FUNCTION_BLOCK FB_Pomp IMPLEMENTS ITF_Pomp
VAR
	InternalToerental : INT; // Internal variable for current speed
 	InternalState : E_PompState;    // Internal variable for pump state
	InternalToerental2 : INT; // Internal variable for current speed
	globaaldoeltoerental : INT; //global variable for doel speed
	
	timeroptoeren : TON;
	timerloopt : BOOL := TRUE;
	optoerentimer : TIME := T#1M;
	
	visvriendelijkactief : BOOL:=visvriendelijkopstartenactief;
	
	//visvriendelijk timer
	timervisvriendelijktijd : TIME := T#3M;
	timervisvriendelijk : TON;
	bezig_visvriendelijkopstarten : BOOL := FALSE;
	
	tagName : STRING;
	outputpompon : ITF_pompdigout;
	inputpompon : ITF_pompdigin;
	outputtoerental : ITF_pompangout;
	
	timerpomperror: ton;
	timerpomperrortijd: TIME:=T#20S;
	noodstop:BOOL;
	
	
	testingbool : bool;
END_VAR

//visvriendelijk
IF visvriendelijkactief AND (StatePomp = E_PompState.off OR bezig_visvriendelijkopstarten) THEN
	bezig_visvriendelijkopstarten:=TRUE;
	visvriendelijk();
END_IF

//outputs pomp
ActueelToerental:=InternalToerental;
outputtoerental.set(InternalToerental);
IF InternalToerental = 0 AND globaaldoeltoerental=0 THEN
	outputpompon.set(FALSE);
ELSIF globaaldoeltoerental>0 THEN
	outputpompon.set(TRUE);
END_IF
testingbool:= inputpompon.get(FALSE);
//inputs errorcheck
timerpomperror(in:=( NOT (inputpompon.get(FALSE)) AND(globaaldoeltoerental>0 AND ActueelToerental>0)) OR(inputpompon.get(TRUE) AND ((InternalToerental = 0 AND globaaldoeltoerental=0) OR ActueelToerental=0)), PT:=timerpomperrortijd);
IF timerpomperror.Q THEN
	InternalState := E_PompState.error;
END_IF

//status pomp
IF (NOT timerpomperror.Q) THEN
	IF  inputpompon.get(FALSE) AND ActueelToerental=0 THEN
		InternalState := E_pompstate.off;
	ELSIF inputpompon.get(TRUE) AND ActueelToerental<globaaldoeltoerental THEN
		InternalState := E_pompstate.optoeren;
	ELSIF inputpompon.get(TRUE) AND ActueelToerental>globaaldoeltoerental THEN
		InternalState := E_pompstate.aftoeren;
	ELSIF inputpompon.get(TRUE) AND ActueelToerental=globaaldoeltoerental THEN
		InternalState := E_pompstate.on;
	END_IF
END_IF

{warning 'Add property implementation'}
PROPERTY ActueelToerental : INT
GET
 ActueelToerental := InternalToerental;
END_GET
SET
    InternalToerental := ActueelToerental;
END_SET
END_PROPERTY

//FB_Init is always available implicitly and it is used primarily for initialization.
//The return value is not evaluated. For a specific influence, you can also declare the
//methods explicitly and provide additional code there with the standard initialization
//code. You can evaluate the return value.
METHOD FB_Init: BOOL
VAR_INPUT
    bInitRetains: BOOL; // TRUE: the retain variables are initialized (reset warm / reset cold)
    bInCopyCode: BOOL;  // TRUE: the instance will be copied to the copy code afterward (online change)   
	tag : STRING;
	DigOutOn : ITF_pompdigout;
	Diginon : ITF_pompdigin;
	Anaouttoerental : ITF_pompangout;
END_VAR
tagname := tag;
outputpompon := DigOutOn;
inputpompon := Diginon;
outputtoerental := Anaouttoerental;
END_METHOD

METHOD PompGoTo : INT
VAR_INPUT
	toerental	: INT;
END_VAR

VAR
	afnametoerental : INT :=20;
	toenamentoerental : INT :=20;
END_VAR
timeroptoeren(IN := timerloopt, PT := optoerentimer);
globaaldoeltoerental:=toerental;
IF noodstop THEN
	InternalToerental:=0;
ELSIF timeroptoeren.Q AND NOT bezig_visvriendelijkopstarten THEN
	timerloopt := FALSE;
	IF (toerental <= InternalToerental+toenamentoerental) AND (toerental >= InternalToerental-afnametoerental) THEN
		IF toerental >20 OR TOERENTAL=0THEN	
		InternalToerental:= toerental;
		ELSIF TOERENTAL>0 THEN
			INTERNALTOERENTAL:=20;
		END_IF;
	ELSIF toerental > InternalToerental THEN
	InternalToerental := InternalToerental+toenamentoerental;
	ELSIF toerental < internaltoerental THEN
		internaltoerental := InternalToerental-afnametoerental;
	END_IF;
ELSE
	timerloopt:=TRUE;
END_IF
END_METHOD

{warning 'Add property implementation'}
PROPERTY StatePomp : E_PompState
GET
    StatePomp := InternalState;
END_GET
SET
    InternalState := StatePomp;
END_SET
END_PROPERTY

METHOD visvriendelijk : BOOL
VAR_INPUT
END_VAR
timervisvriendelijk(IN:= bezig_visvriendelijkopstarten, PT:= timervisvriendelijktijd);

IF timervisvriendelijk.Q THEN
	bezig_visvriendelijkopstarten:=FALSE;
ELSE
	InternalToerental:=20;
END_IF
END_METHOD

PROPERTY visvriendelijkopstartenactief : bool
GET
visvriendelijkopstartenactief:=visvriendelijkactief;
END_GET
SET
visvriendelijkactief:=visvriendelijkopstartenactief;
END_SET
END_PROPERTY

END_FUNCTION_BLOCK

(* stored: Version 1.1.0.1, ProductVersion 3.1.4026.8
   POU FB_Pomp: Id {01e0e1ca-9203-401d-bd28-bd8ab180b19f}, SpecialFunc None
   Property ActueelToerental: Id {88d60577-962c-4c2d-820d-3c715054a2e6}
   Get Get: Id {6ce3d73e-f992-458e-b779-47ddd6581a09}
   Set Set: Id {3edb9cc8-aede-44bb-a200-c22dffcdef8b}
   Method FB_Init: Id {dc539e09-6f97-4e59-8bee-fe04507eedbf}
   Method PompGoTo: Id {0c4c33cf-85bb-4137-9363-b61f6c82564a}
   Property StatePomp: Id {a3356c66-7303-4084-af63-de2a393bc632}
   Get Get: Id {41be7f56-846c-4dde-9931-f12128d4dd95}
   Set Set: Id {515ac4c7-2fb1-4d81-bf82-c7c0bb4a75f9}
   Method visvriendelijk: Id {816aedc3-4076-4bc8-9819-9e22edb44f46}
   Property visvriendelijkopstartenactief: Id {18bd2c40-b027-4d2f-96e2-b7d1f3444e47}
   Get Get: Id {51de95b2-8432-4e7e-9c4e-3e03cf6d5873}
   Set Set: Id {1179243f-ab2f-4ad9-afcf-5189fe1266ba} *)
